{attribute 'qualified_only'}
{attribute 'strict'}
{attribute 'to_string'}
TYPE E_MachineCommand :
(
    STOP,
    START
);
END_TYPE

(* stored: Version 1.1.0.1
   DUT E_MachineCommand: Id {02ced208-e2a7-49b5-a892-3b348e3c536e} *)
